INTERFACE I_OutputPortAddedEvent extends I_Event

PROPERTY PUBLIC Target : I_OutputPort
GET
END_GET
END_PROPERTY

END_INTERFACE

(* stored: Version 1.1.0.1, ProductVersion 3.1.4024.12
   Itf I_OutputPortAddedEvent: Id {2ba242a2-35d9-488d-b10e-19a4c1a80baf}
   Property Target: Id {26c70837-32f4-4e60-b2ef-d1a9b3644f1d}
   Get Get: Id {1d4c2356-bd7f-4290-95fa-87d0011505d2} *)
